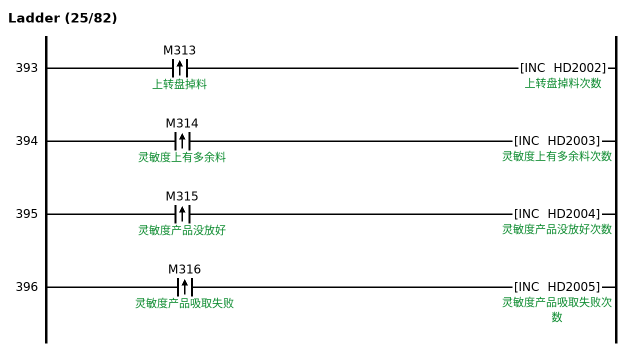
[picture p24: Ladder rows 393-396]
LDP    M313	; 上转盘掉料
INC    HD2002	; 上转盘掉料次数
LDP    M314	; 灵敏度上有多余料
INC    HD2003	; 灵敏度上有多余料次数
LDP    M315	; 灵敏度产品没放好
INC    HD2004	; 灵敏度产品没放好次数
LDP    M316	; 灵敏度产品吸取失败
INC    HD2005	; 灵敏度产品吸取失败次数

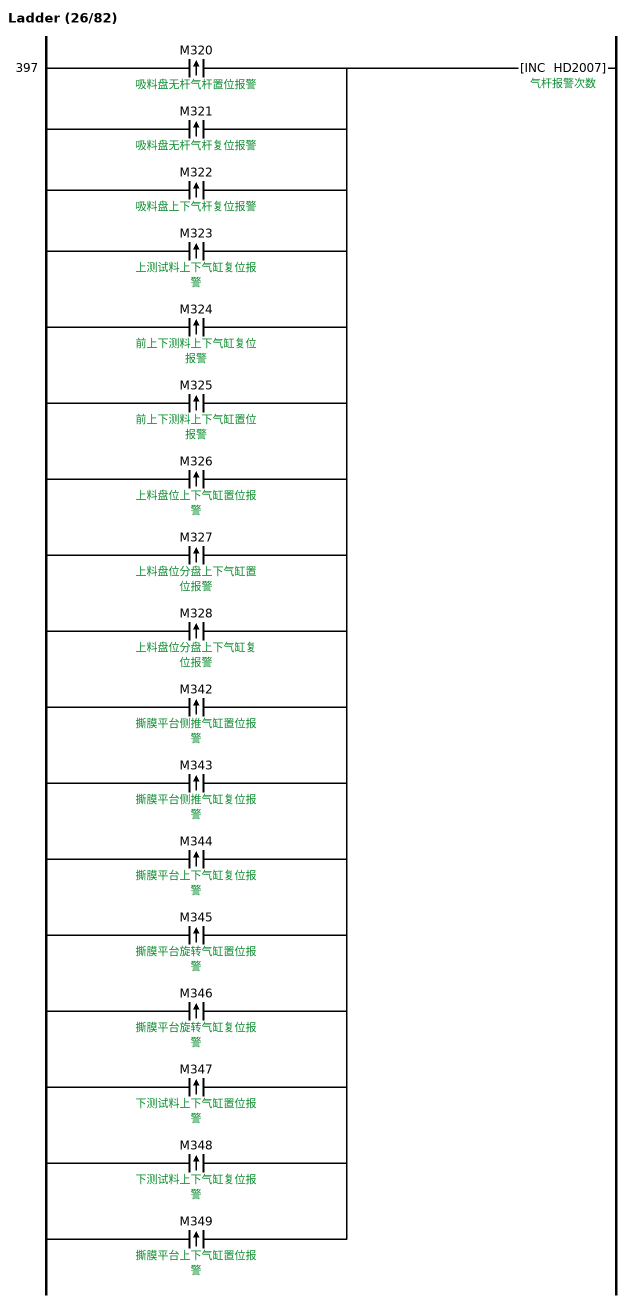
LDP    M320	; 吸料盘无杆气杆置位报警
ORP    M321	; 吸料盘无杆气杆复位报警
ORP    M322	; 吸料盘上下气杆复位报警
ORP    M323	; 上测试料上下气缸复位报警
ORP    M324	; 前上下测料上下气缸复位报警
ORP    M325	; 前上下测料上下气缸置位报警
ORP    M326	; 上料盘位上下气缸置位报警
ORP    M327	; 上料盘位分盘上下气缸置位报警
ORP    M328	; 上料盘位分盘上下气缸复位报警
ORP    M342	; 撕膜平台侧推气缸置位报警
ORP    M343	; 撕膜平台侧推气缸复位报警
ORP    M344	; 撕膜平台上下气缸复位报警
ORP    M345	; 撕膜平台旋转气缸置位报警
ORP    M346	; 撕膜平台旋转气缸复位报警
ORP    M347	; 下测试料上下气缸置位报警
ORP    M348	; 下测试料上下气缸复位报警
ORP    M349	; 撕膜平台上下气缸置位报警
INC    HD2007	; 气杆报警次数

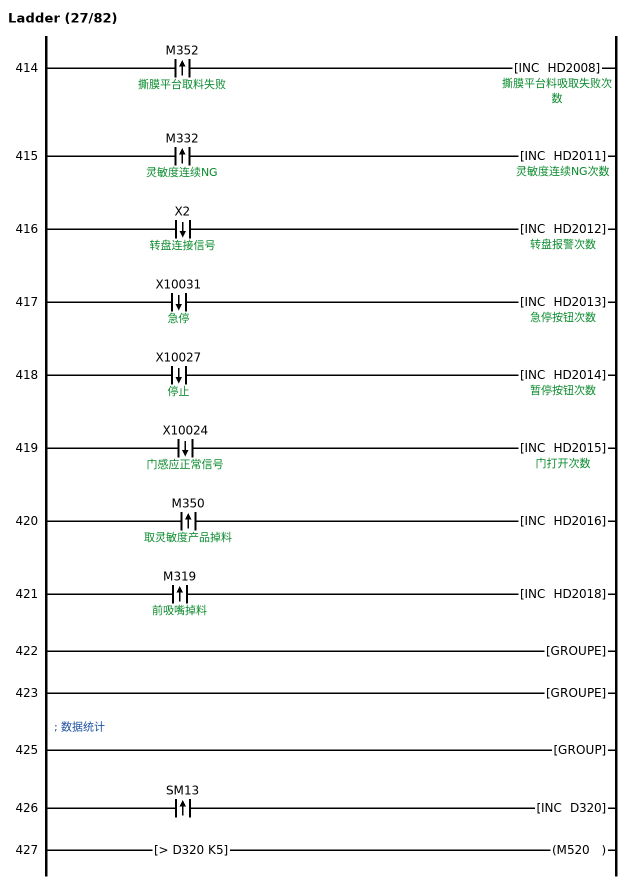
LDP    M352	; 撕膜平台取料失败
INC    HD2008	; 撕膜平台料吸取失败次数
LDP    M332	; 灵敏度连续NG
INC    HD2011	; 灵敏度连续NG次数
LDF    X2	; 转盘连接信号
INC    HD2012	; 转盘报警次数
LDF    X10031	; 急停
INC    HD2013	; 急停按钮次数
LDF    X10027	; 停止
INC    HD2014	; 暂停按钮次数
LDF    X10024	; 门感应正常信号
INC    HD2015	; 门打开次数
LDP    M350	; 取灵敏度产品掉料
INC    HD2016
LDP    M319	; 前吸嘴掉料
INC    HD2018
GROUPE
GROUPE
; 数据统计
GROUP
LDP    SM13
INC    D320
LD>    D320 K5
OUT    M520

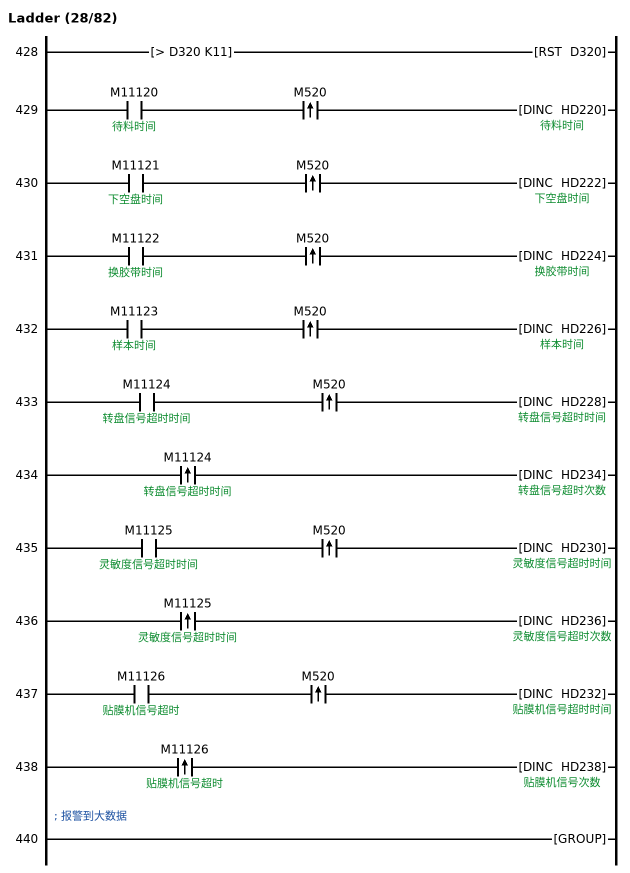
LD>    D320 K11
RST    D320
LD     M11120	; 待料时间
ANDP   M520
DINC   HD220	; 待料时间
LD     M11121	; 下空盘时间
ANDP   M520
DINC   HD222	; 下空盘时间
LD     M11122	; 换胶带时间
ANDP   M520
DINC   HD224	; 换胶带时间
LD     M11123	; 样本时间
ANDP   M520
DINC   HD226	; 样本时间
LD     M11124	; 转盘信号超时时间
ANDP   M520
DINC   HD228	; 转盘信号超时时间
LDP    M11124	; 转盘信号超时时间
DINC   HD234	; 转盘信号超时次数
LD     M11125	; 灵敏度信号超时时间
ANDP   M520
DINC   HD230	; 灵敏度信号超时时间
LDP    M11125	; 灵敏度信号超时时间
DINC   HD236	; 灵敏度信号超时次数
LD     M11126	; 贴膜机信号超时
ANDP   M520
DINC   HD232	; 贴膜机信号超时时间
LDP    M11126	; 贴膜机信号超时
DINC   HD238	; 贴膜机信号次数
; 报警到大数据
GROUP

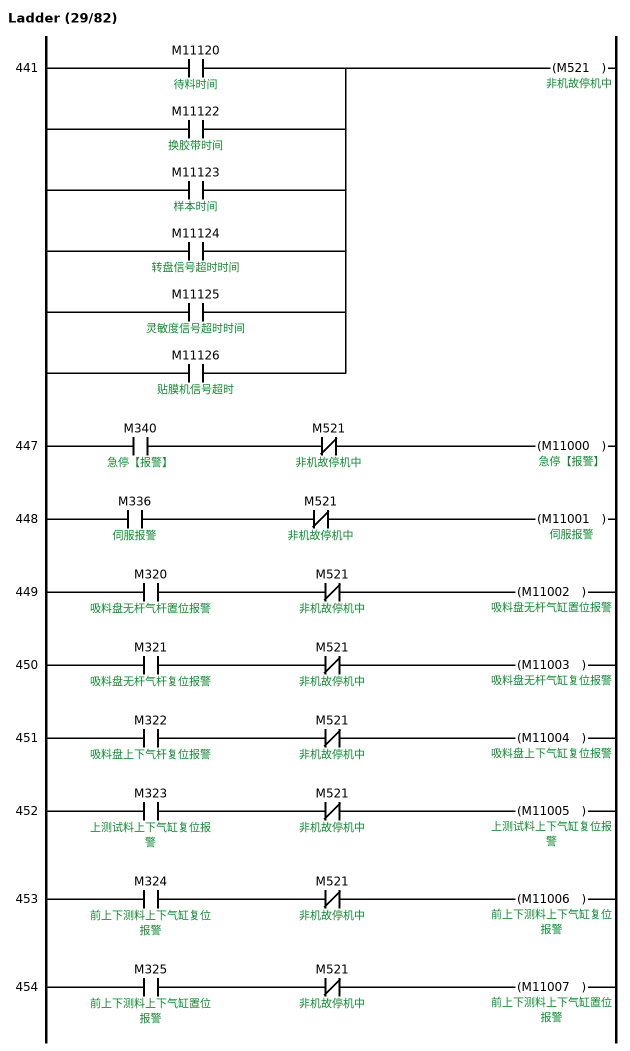
LD     M11120	; 待料时间
OR     M11122	; 换胶带时间
OR     M11123	; 样本时间
OR     M11124	; 转盘信号超时时间
OR     M11125	; 灵敏度信号超时时间
OR     M11126	; 贴膜机信号超时
OUT    M521	; 非机故停机中
LD     M340	; 急停【报警】
ANI    M521	; 非机故停机中
OUT    M11000	; 急停【报警】
LD     M336	; 伺服报警
ANI    M521	; 非机故停机中
OUT    M11001	; 伺服报警
LD     M320	; 吸料盘无杆气杆置位报警
ANI    M521	; 非机故停机中
OUT    M11002	; 吸料盘无杆气缸置位报警
LD     M321	; 吸料盘无杆气杆复位报警
ANI    M521	; 非机故停机中
OUT    M11003	; 吸料盘无杆气缸复位报警
LD     M322	; 吸料盘上下气杆复位报警
ANI    M521	; 非机故停机中
OUT    M11004	; 吸料盘上下气缸复位报警
LD     M323	; 上测试料上下气缸复位报警
ANI    M521	; 非机故停机中
OUT    M11005	; 上测试料上下气缸复位报警
LD     M324	; 前上下测料上下气缸复位报警
ANI    M521	; 非机故停机中
OUT    M11006	; 前上下测料上下气缸复位报警
LD     M325	; 前上下测料上下气缸置位报警
ANI    M521	; 非机故停机中
OUT    M11007	; 前上下测料上下气缸置位报警

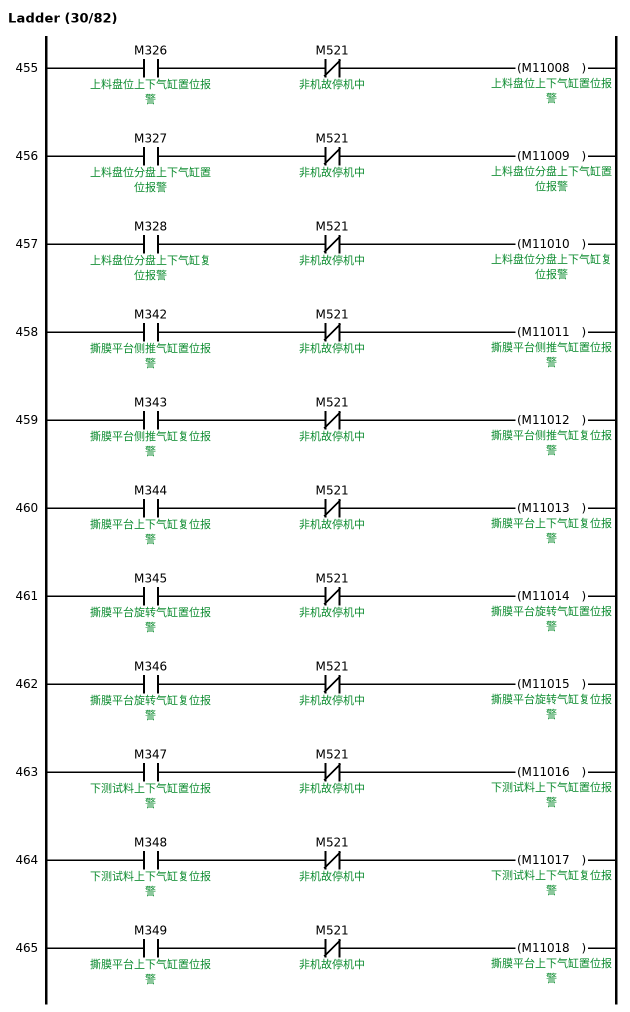
LD     M326	; 上料盘位上下气缸置位报警
ANI    M521	; 非机故停机中
OUT    M11008	; 上料盘位上下气缸置位报警
LD     M327	; 上料盘位分盘上下气缸置位报警
ANI    M521	; 非机故停机中
OUT    M11009	; 上料盘位分盘上下气缸置位报警
LD     M328	; 上料盘位分盘上下气缸复位报警
ANI    M521	; 非机故停机中
OUT    M11010	; 上料盘位分盘上下气缸复位报警
LD     M342	; 撕膜平台侧推气缸置位报警
ANI    M521	; 非机故停机中
OUT    M11011	; 撕膜平台侧推气缸置位报警
LD     M343	; 撕膜平台侧推气缸复位报警
ANI    M521	; 非机故停机中
OUT    M11012	; 撕膜平台侧推气缸复位报警
LD     M344	; 撕膜平台上下气缸复位报警
ANI    M521	; 非机故停机中
OUT    M11013	; 撕膜平台上下气缸复位报警
LD     M345	; 撕膜平台旋转气缸置位报警
ANI    M521	; 非机故停机中
OUT    M11014	; 撕膜平台旋转气缸置位报警
LD     M346	; 撕膜平台旋转气缸复位报警
ANI    M521	; 非机故停机中
OUT    M11015	; 撕膜平台旋转气缸复位报警
LD     M347	; 下测试料上下气缸置位报警
ANI    M521	; 非机故停机中
OUT    M11016	; 下测试料上下气缸置位报警
LD     M348	; 下测试料上下气缸复位报警
ANI    M521	; 非机故停机中
OUT    M11017	; 下测试料上下气缸复位报警
LD     M349	; 撕膜平台上下气缸置位报警
ANI    M521	; 非机故停机中
OUT    M11018	; 撕膜平台上下气缸置位报警

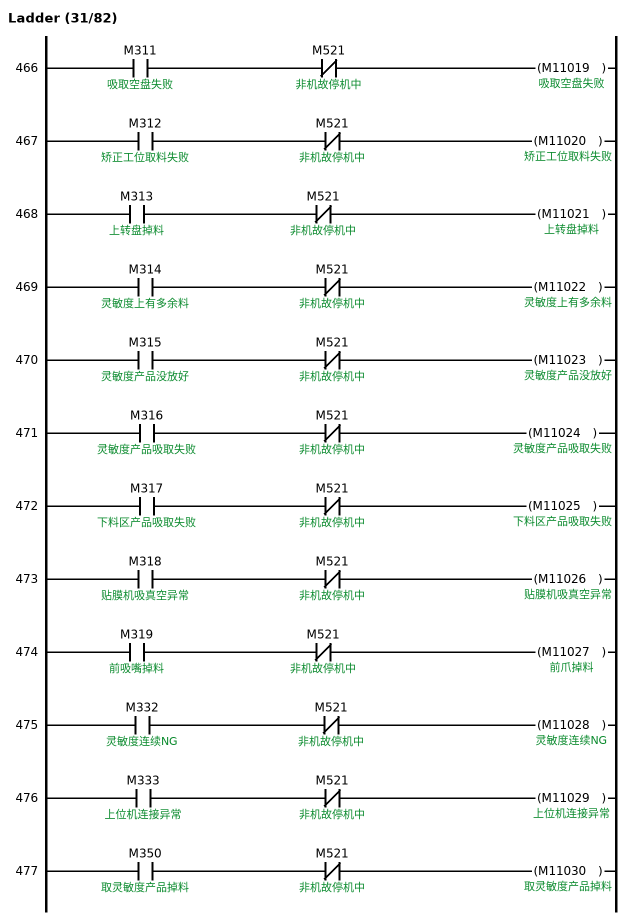
LD     M311	; 吸取空盘失败
ANI    M521	; 非机故停机中
OUT    M11019	; 吸取空盘失败
LD     M312	; 矫正工位取料失败
ANI    M521	; 非机故停机中
OUT    M11020	; 矫正工位取料失败
LD     M313	; 上转盘掉料
ANI    M521	; 非机故停机中
OUT    M11021	; 上转盘掉料
LD     M314	; 灵敏度上有多余料
ANI    M521	; 非机故停机中
OUT    M11022	; 灵敏度上有多余料
LD     M315	; 灵敏度产品没放好
ANI    M521	; 非机故停机中
OUT    M11023	; 灵敏度产品没放好
LD     M316	; 灵敏度产品吸取失败
ANI    M521	; 非机故停机中
OUT    M11024	; 灵敏度产品吸取失败
LD     M317	; 下料区产品吸取失败
ANI    M521	; 非机故停机中
OUT    M11025	; 下料区产品吸取失败
LD     M318	; 贴膜机吸真空异常
ANI    M521	; 非机故停机中
OUT    M11026	; 贴膜机吸真空异常
LD     M319	; 前吸嘴掉料
ANI    M521	; 非机故停机中
OUT    M11027	; 前爪掉料
LD     M332	; 灵敏度连续NG
ANI    M521	; 非机故停机中
OUT    M11028	; 灵敏度连续NG
LD     M333	; 上位机连接异常
ANI    M521	; 非机故停机中
OUT    M11029	; 上位机连接异常
LD     M350	; 取灵敏度产品掉料
ANI    M521	; 非机故停机中
OUT    M11030	; 取灵敏度产品掉料

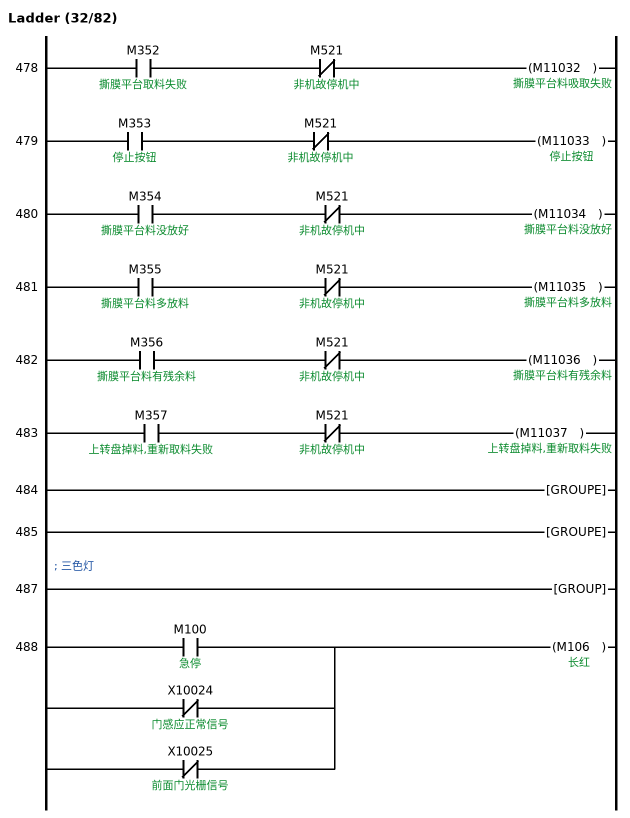
LD     M352	; 撕膜平台取料失败
ANI    M521	; 非机故停机中
OUT    M11032	; 撕膜平台料吸取失败
LD     M353	; 停止按钮
ANI    M521	; 非机故停机中
OUT    M11033	; 停止按钮
LD     M354	; 撕膜平台料没放好
ANI    M521	; 非机故停机中
OUT    M11034	; 撕膜平台料没放好
LD     M355	; 撕膜平台料多放料
ANI    M521	; 非机故停机中
OUT    M11035	; 撕膜平台料多放料
LD     M356	; 撕膜平台料有残余料
ANI    M521	; 非机故停机中
OUT    M11036	; 撕膜平台料有残余料
LD     M357	; 上转盘掉料,重新取料失败
ANI    M521	; 非机故停机中
OUT    M11037	; 上转盘掉料,重新取料失败
GROUPE
GROUPE
; 三色灯
GROUP
LD     M100	; 急停
ORI    X10024	; 门感应正常信号
ORI    X10025	; 前面门光栅信号
OUT    M106	; 长红

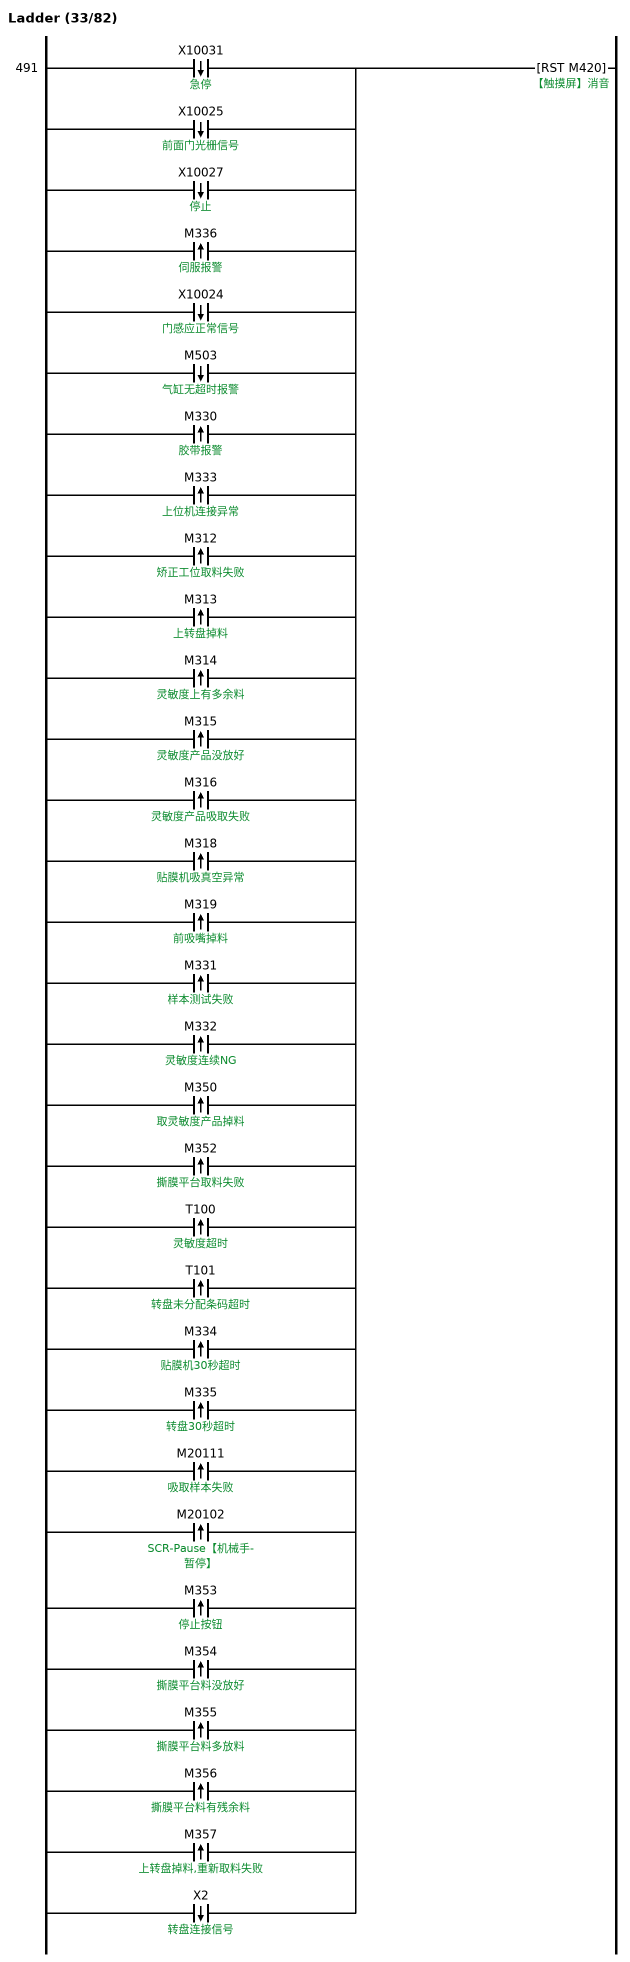
LDF    X10031	; 急停
ORF    X10025	; 前面门光栅信号
ORF    X10027	; 停止
ORP    M336	; 伺服报警
ORF    X10024	; 门感应正常信号
ORF    M503	; 气缸无超时报警
ORP    M330	; 胶带报警
ORP    M333	; 上位机连接异常
ORP    M312	; 矫正工位取料失败
ORP    M313	; 上转盘掉料
ORP    M314	; 灵敏度上有多余料
ORP    M315	; 灵敏度产品没放好
ORP    M316	; 灵敏度产品吸取失败
ORP    M318	; 贴膜机吸真空异常
ORP    M319	; 前吸嘴掉料
ORP    M331	; 样本测试失败
ORP    M332	; 灵敏度连续NG
ORP    M350	; 取灵敏度产品掉料
ORP    M352	; 撕膜平台取料失败
ORP    T100	; 灵敏度超时
ORP    T101	; 转盘未分配条码超时
ORP    M334	; 贴膜机30秒超时
ORP    M335	; 转盘30秒超时
ORP    M20111	; 吸取样本失败
ORP    M20102	; SCR-Pause【机械手-暂停】
ORP    M353	; 停止按钮
ORP    M354	; 撕膜平台料没放好
ORP    M355	; 撕膜平台料多放料
ORP    M356	; 撕膜平台料有残余料
ORP    M357	; 上转盘掉料,重新取料失败
ORF    X2	; 转盘连接信号
RST    M420	; 【触摸屏】消音

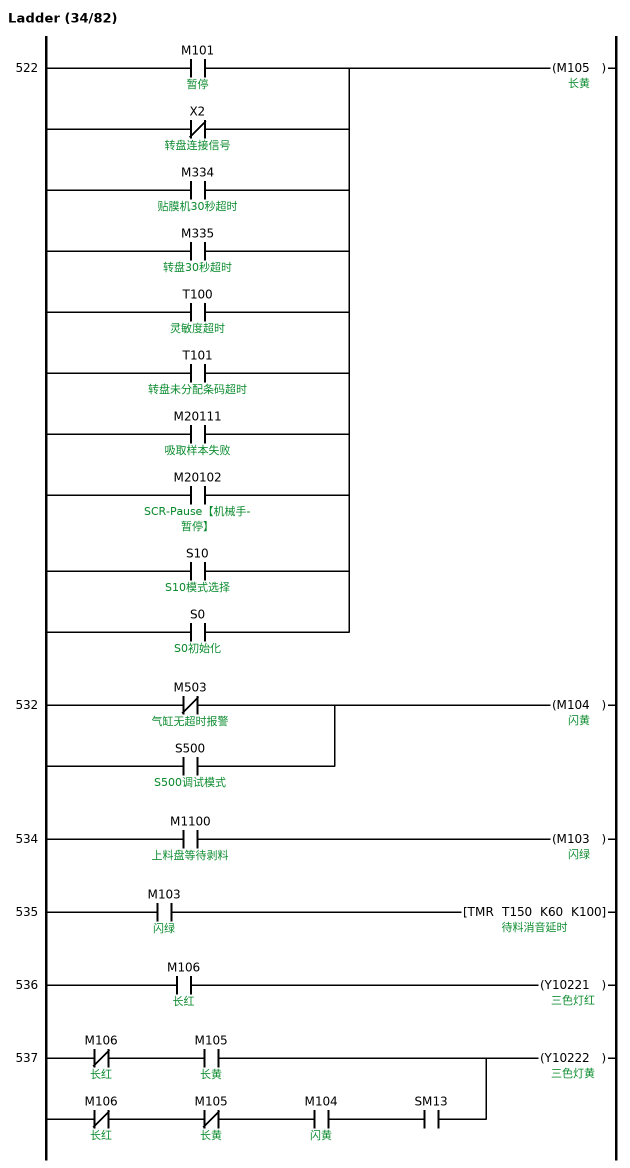
LD     M101	; 暂停
ORI    X2	; 转盘连接信号
OR     M334	; 贴膜机30秒超时
OR     M335	; 转盘30秒超时
OR     T100	; 灵敏度超时
OR     T101	; 转盘未分配条码超时
OR     M20111	; 吸取样本失败
OR     M20102	; SCR-Pause【机械手-暂停】
OR     S10	; S10模式选择
OR     S0	; S0初始化
OUT    M105	; 长黄
LDI    M503	; 气缸无超时报警
OR     S500	; S500调试模式
OUT    M104	; 闪黄
LD     M1100	; 上料盘等待剥料
OUT    M103	; 闪绿
LD     M103	; 闪绿
TMR    T150 K60 K100	; 待料消音延时
LD     M106	; 长红
OUT    Y10221	; 三色灯红
LDI    M106	; 长红
AND    M105	; 长黄
LDI    M106	; 长红
ANI    M105	; 长黄
AND    M104	; 闪黄
AND    SM13
ORB
OUT    Y10222	; 三色灯黄

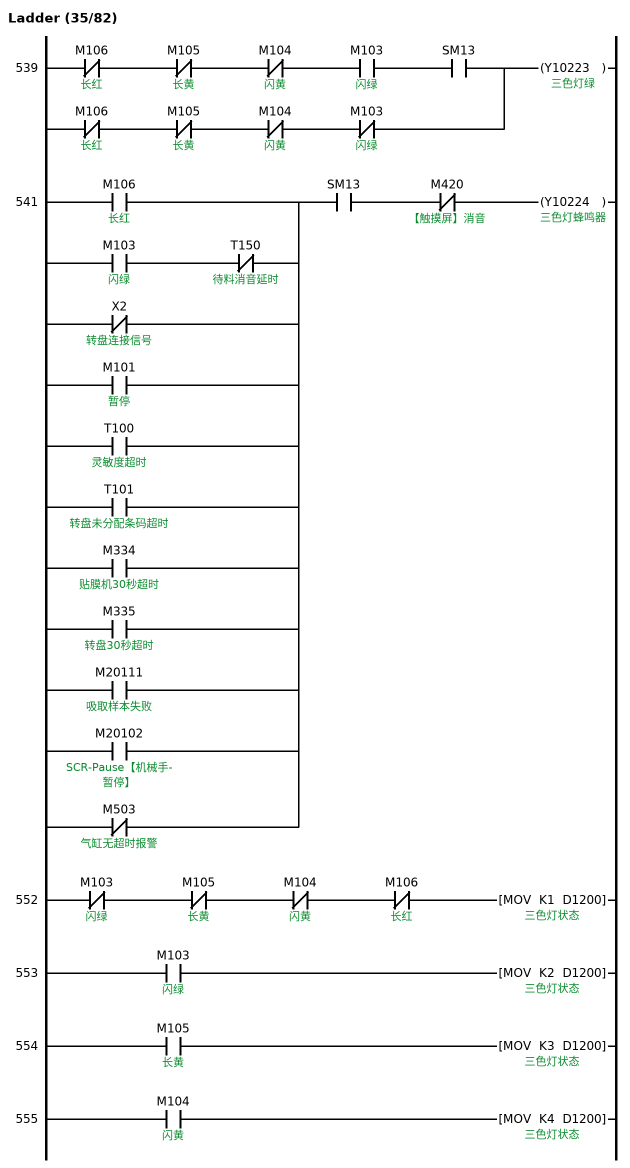
LDI    M106	; 长红
ANI    M105	; 长黄
ANI    M104	; 闪黄
AND    M103	; 闪绿
AND    SM13
LDI    M106	; 长红
ANI    M105	; 长黄
ANI    M104	; 闪黄
ANI    M103	; 闪绿
ORB
OUT    Y10223	; 三色灯绿
LD     M106	; 长红
LD     M103	; 闪绿
ANI    T150	; 待料消音延时
ORB
ORI    X2	; 转盘连接信号
OR     M101	; 暂停
OR     T100	; 灵敏度超时
OR     T101	; 转盘未分配条码超时
OR     M334	; 贴膜机30秒超时
OR     M335	; 转盘30秒超时
OR     M20111	; 吸取样本失败
OR     M20102	; SCR-Pause【机械手-暂停】
ORI    M503	; 气缸无超时报警
AND    SM13
ANI    M420	; 【触摸屏】消音
OUT    Y10224	; 三色灯蜂鸣器
LDI    M103	; 闪绿
ANI    M105	; 长黄
ANI    M104	; 闪黄
ANI    M106	; 长红
MOV    K1 D1200	; 三色灯状态
LD     M103	; 闪绿
MOV    K2 D1200	; 三色灯状态
LD     M105	; 长黄
MOV    K3 D1200	; 三色灯状态
LD     M104	; 闪黄
MOV    K4 D1200	; 三色灯状态

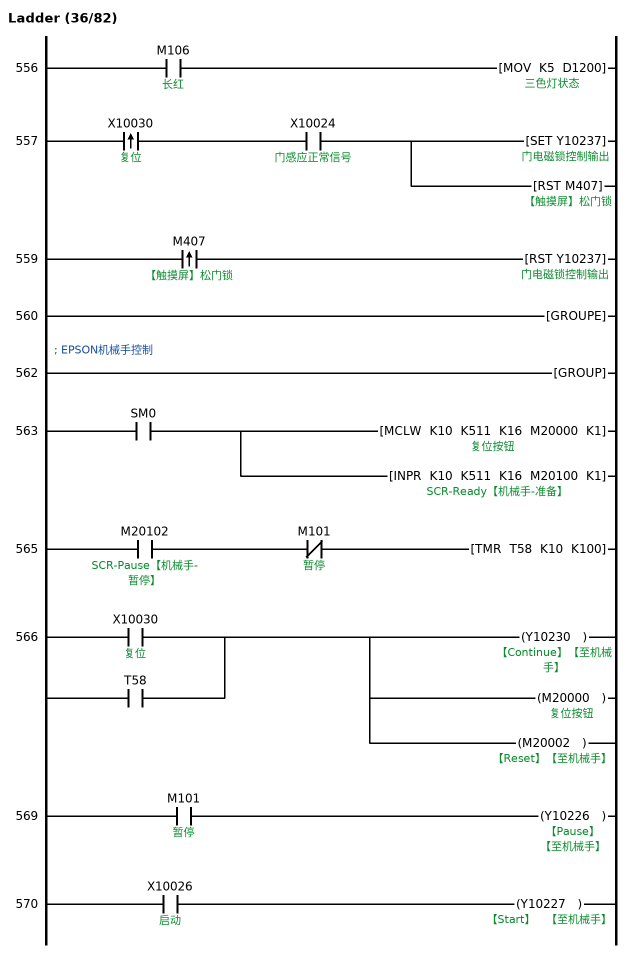
LD     M106	; 长红
MOV    K5 D1200	; 三色灯状态
LDP    X10030	; 复位
AND    X10024	; 门感应正常信号
SET    Y10237	; 门电磁锁控制输出
RST    M407	; 【触摸屏】松门锁
LDP    M407	; 【触摸屏】松门锁
RST    Y10237	; 门电磁锁控制输出
GROUPE
; EPSON机械手控制
GROUP
LD     SM0
MCLW   K10 K511 K16 M20000 K1	; 复位按钮
INPR   K10 K511 K16 M20100 K1	; SCR-Ready【机械手-准备】
LD     M20102	; SCR-Pause【机械手-暂停】
ANI    M101	; 暂停
TMR    T58 K10 K100
LD     X10030	; 复位
OR     T58
OUT    Y10230	; 【Continue】【至机械手】
OUT    M20000	; 复位按钮
OUT    M20002	; 【Reset】【至机械手】
LD     M101	; 暂停
OUT    Y10226	; 【Pause】   【至机械手】
LD     X10026	; 启动
OUT    Y10227	; 【Start】   【至机械手】

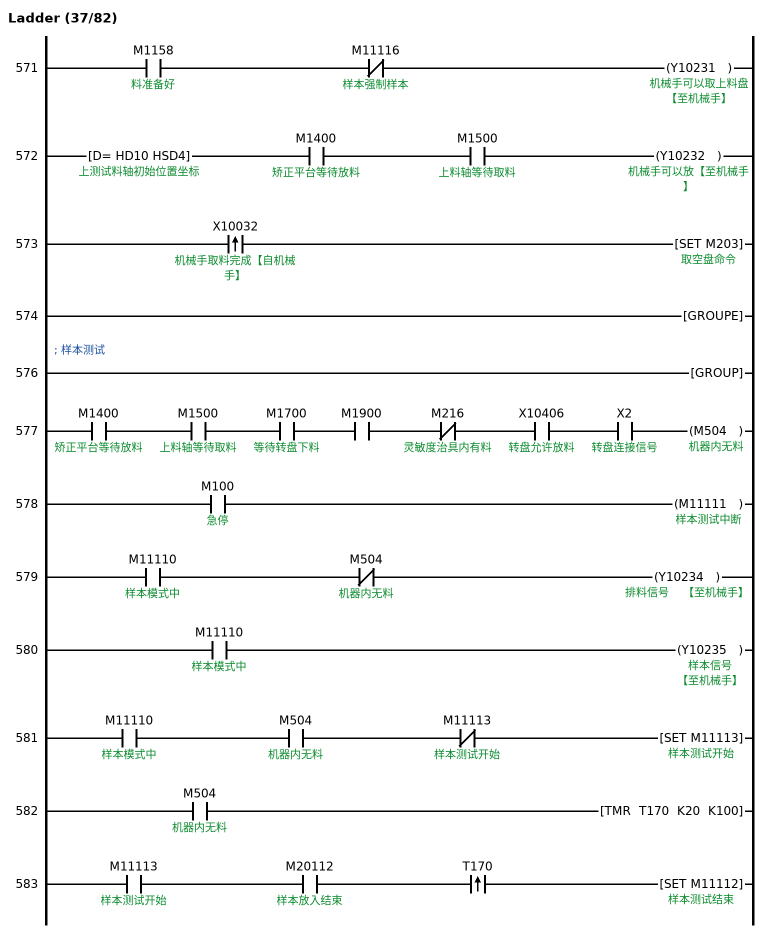
LD     M1158	; 料准备好
ANI    M11116	; 样本强制样本
OUT    Y10231	; 机械手可以取上料盘  【至机械手】
DLD=   HD10 HSD4	; 上测试料轴初始位置坐标
AND    M1400	; 矫正平台等待放料
AND    M1500	; 上料轴等待取料
OUT    Y10232	; 机械手可以放【至机械手】
LDP    X10032	; 机械手取料完成【自机械手】
SET    M203	; 取空盘命令
GROUPE
; 样本测试
GROUP
LD     M1400	; 矫正平台等待放料
AND    M1500	; 上料轴等待取料
AND    M1700	; 等待转盘下料
AND    M1900
ANI    M216	; 灵敏度治具内有料
AND    X10406	; 转盘允许放料
AND    X2	; 转盘连接信号
OUT    M504	; 机器内无料
LD     M100	; 急停
OUT    M11111	; 样本测试中断
LD     M11110	; 样本模式中
ANI    M504	; 机器内无料
OUT    Y10234	; 排料信号    【至机械手】
LD     M11110	; 样本模式中
OUT    Y10235	; 样本信号     【至机械手】
LD     M11110	; 样本模式中
AND    M504	; 机器内无料
ANI    M11113	; 样本测试开始
SET    M11113	; 样本测试开始
LD     M504	; 机器内无料
TMR    T170 K20 K100
LD     M11113	; 样本测试开始
AND    M20112	; 样本放入结束
ANDP   T170
SET    M11112	; 样本测试结束

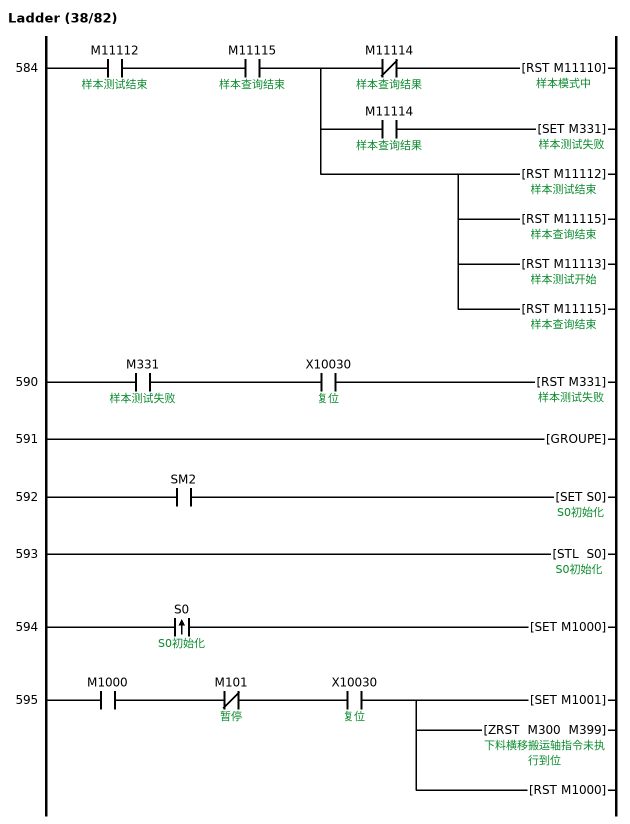
LD     M11112	; 样本测试结束
AND    M11115	; 样本查询结束
MPS
ANI    M11114	; 样本查询结果
RST    M11110	; 样本模式中
MRD
AND    M11114	; 样本查询结果
SET    M331	; 样本测试失败
MPP
RST    M11112	; 样本测试结束
RST    M11115	; 样本查询结束
RST    M11113	; 样本测试开始
RST    M11115	; 样本查询结束
LD     M331	; 样本测试失败
AND    X10030	; 复位
RST    M331	; 样本测试失败
GROUPE
LD     SM2
SET    S0	; S0初始化
STL    S0	; S0初始化
LDP    S0	; S0初始化
SET    M1000
LD     M1000
ANI    M101	; 暂停
AND    X10030	; 复位
SET    M1001
ZRST   M300 M399	; 下料横移搬运轴指令未执行到位
RST    M1000

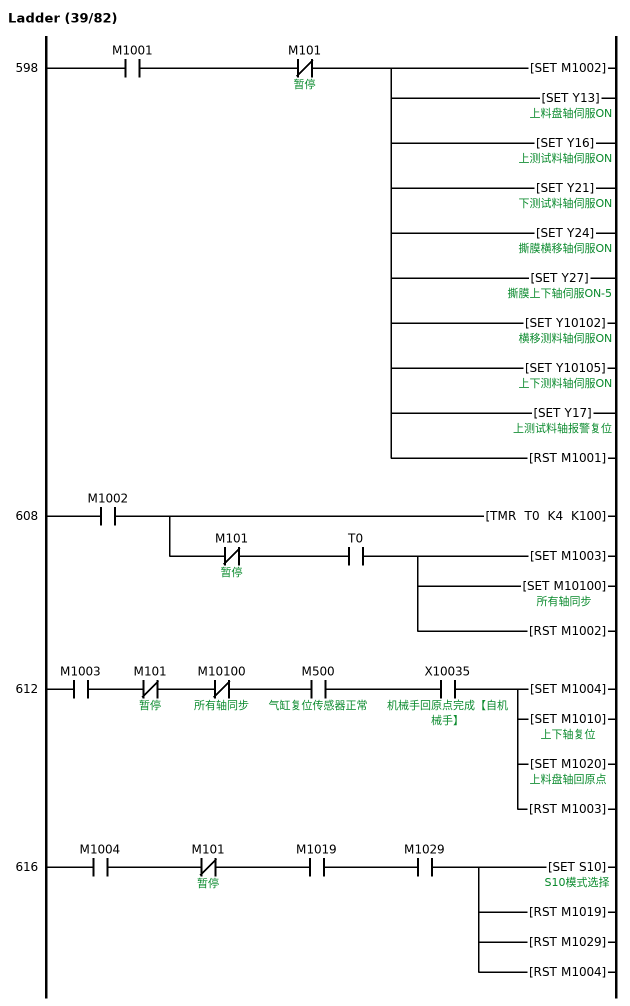
LD     M1001
ANI    M101	; 暂停
SET    M1002
SET    Y13	; 上料盘轴伺服ON
SET    Y16	; 上测试料轴伺服ON
SET    Y21	; 下测试料轴伺服ON
SET    Y24	; 撕膜横移轴伺服ON
SET    Y27	; 撕膜上下轴伺服ON-5
SET    Y10102	; 横移测料轴伺服ON
SET    Y10105	; 上下测料轴伺服ON
SET    Y17	; 上测试料轴报警复位
RST    M1001
LD     M1002
TMR    T0 K4 K100
ANI    M101	; 暂停
AND    T0
SET    M1003
SET    M10100	; 所有轴同步
RST    M1002
LD     M1003
ANI    M101	; 暂停
ANI    M10100	; 所有轴同步
AND    M500	; 气缸复位传感器正常
AND    X10035	; 机械手回原点完成【自机械手】
SET    M1004
SET    M1010	; 上下轴复位
SET    M1020	; 上料盘轴回原点
RST    M1003
LD     M1004
ANI    M101	; 暂停
AND    M1019
AND    M1029
SET    S10	; S10模式选择
RST    M1019
RST    M1029
RST    M1004

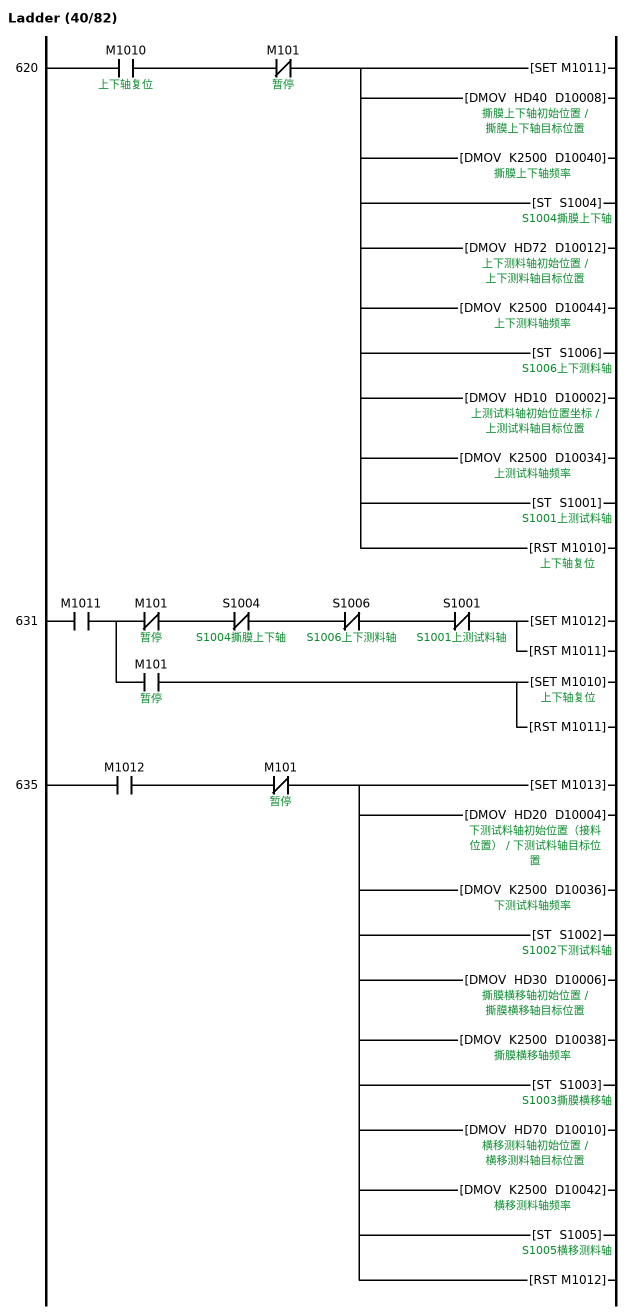
LD     M1010	; 上下轴复位
ANI    M101	; 暂停
SET    M1011
DMOV   HD40 D10008	; 撕膜上下轴初始位置 / 撕膜上下轴目标位置
DMOV   K2500 D10040	; 撕膜上下轴频率
ST     S1004	; S1004撕膜上下轴
DMOV   HD72 D10012	; 上下测料轴初始位置 / 上下测料轴目标位置
DMOV   K2500 D10044	; 上下测料轴频率
ST     S1006	; S1006上下测料轴
DMOV   HD10 D10002	; 上测试料轴初始位置坐标 / 上测试料轴目标位置
DMOV   K2500 D10034	; 上测试料轴频率
ST     S1001	; S1001上测试料轴
RST    M1010	; 上下轴复位
LD     M1011
MPS
ANI    M101	; 暂停
ANI    S1004	; S1004撕膜上下轴
ANI    S1006	; S1006上下测料轴
ANI    S1001	; S1001上测试料轴
SET    M1012
RST    M1011
MPP
AND    M101	; 暂停
SET    M1010	; 上下轴复位
RST    M1011
LD     M1012
ANI    M101	; 暂停
SET    M1013
DMOV   HD20 D10004	; 下测试料轴初始位置（接料位置） / 下测试料轴目标位置
DMOV   K2500 D10036	; 下测试料轴频率
ST     S1002	; S1002下测试料轴
DMOV   HD30 D10006	; 撕膜横移轴初始位置 / 撕膜横移轴目标位置
DMOV   K2500 D10038	; 撕膜横移轴频率
ST     S1003	; S1003撕膜横移轴
DMOV   HD70 D10010	; 横移测料轴初始位置 / 横移测料轴目标位置
DMOV   K2500 D10042	; 横移测料轴频率
ST     S1005	; S1005横移测料轴
RST    M1012

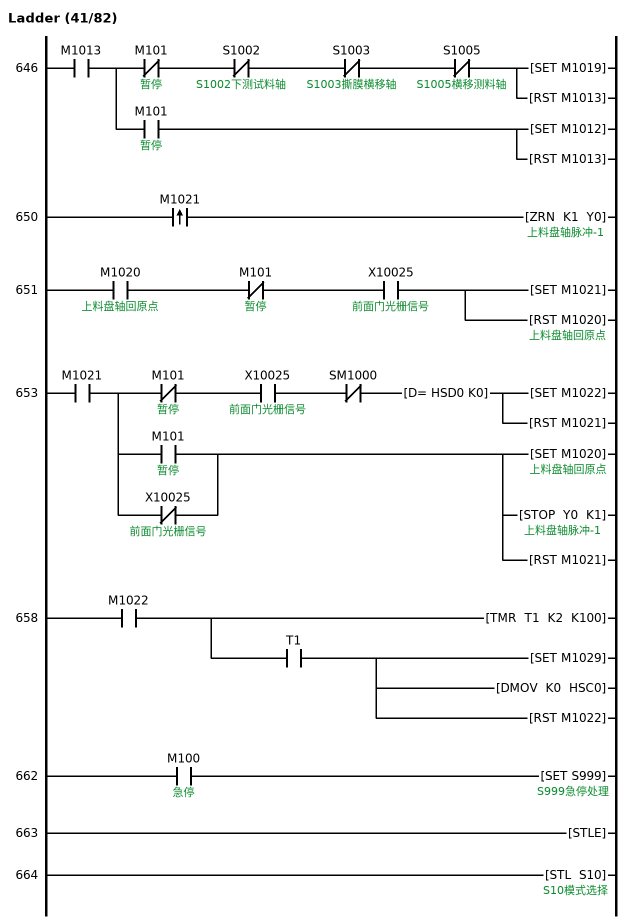
LD     M1013
MPS
ANI    M101	; 暂停
ANI    S1002	; S1002下测试料轴
ANI    S1003	; S1003撕膜横移轴
ANI    S1005	; S1005横移测料轴
SET    M1019
RST    M1013
MPP
AND    M101	; 暂停
SET    M1012
RST    M1013
LDP    M1021
ZRN    K1 Y0	; 上料盘轴脉冲-1
LD     M1020	; 上料盘轴回原点
ANI    M101	; 暂停
AND    X10025	; 前面门光栅信号
SET    M1021
RST    M1020	; 上料盘轴回原点
LD     M1021
MPS
ANI    M101	; 暂停
AND    X10025	; 前面门光栅信号
ANI    SM1000
DAND=  HSD0 K0
SET    M1022
RST    M1021
MPP
LD     M101	; 暂停
ORI    X10025	; 前面门光栅信号
ANB
SET    M1020	; 上料盘轴回原点
STOP   Y0 K1	; 上料盘轴脉冲-1
RST    M1021
LD     M1022
TMR    T1 K2 K100
AND    T1
SET    M1029
DMOV   K0 HSC0
RST    M1022
LD     M100	; 急停
SET    S999	; S999急停处理
STLE
STL    S10	; S10模式选择

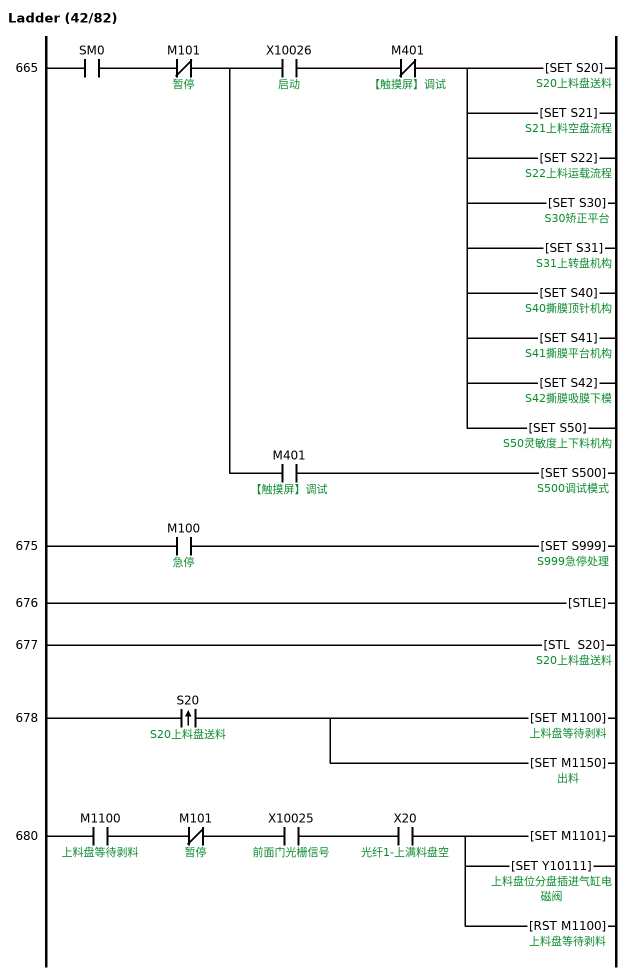
LD     SM0
ANI    M101	; 暂停
MPS
AND    X10026	; 启动
ANI    M401	; 【触摸屏】调试
SET    S20	; S20上料盘送料
SET    S21	; S21上料空盘流程
SET    S22	; S22上料运载流程
SET    S30	; S30矫正平台
SET    S31	; S31上转盘机构
SET    S40	; S40撕膜顶针机构
SET    S41	; S41撕膜平台机构
SET    S42	; S42撕膜吸膜下模
SET    S50	; S50灵敏度上下料机构
MPP
AND    M401	; 【触摸屏】调试
SET    S500	; S500调试模式
LD     M100	; 急停
SET    S999	; S999急停处理
STLE
STL    S20	; S20上料盘送料
LDP    S20	; S20上料盘送料
SET    M1100	; 上料盘等待剥料
SET    M1150	; 出料
LD     M1100	; 上料盘等待剥料
ANI    M101	; 暂停
AND    X10025	; 前面门光栅信号
AND    X20	; 光纤1-上满料盘空
SET    M1101
SET    Y10111	; 上料盘位分盘插进气缸电磁阀
RST    M1100	; 上料盘等待剥料

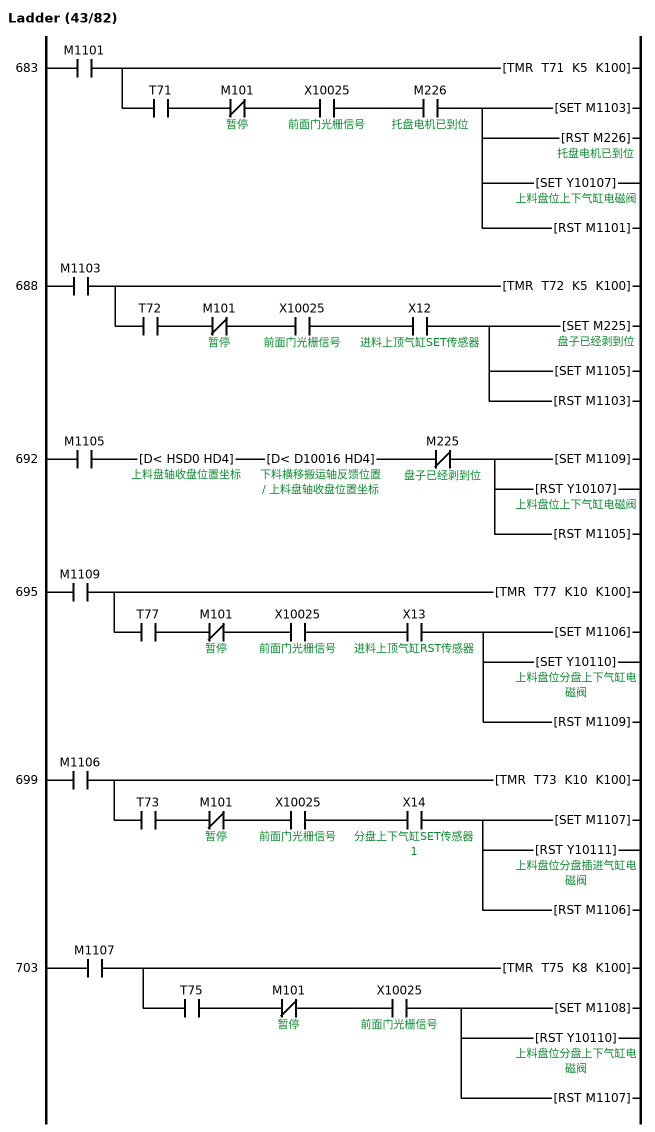
LD     M1101
TMR    T71 K5 K100
AND    T71
ANI    M101	; 暂停
AND    X10025	; 前面门光栅信号
AND    M226	; 托盘电机已到位
SET    M1103
RST    M226	; 托盘电机已到位
SET    Y10107	; 上料盘位上下气缸电磁阀
RST    M1101
LD     M1103
TMR    T72 K5 K100
AND    T72
ANI    M101	; 暂停
AND    X10025	; 前面门光栅信号
AND    X12	; 进料上顶气缸SET传感器
SET    M225	; 盘子已经剥到位
SET    M1105
RST    M1103
LD     M1105
DAND<  HSD0 HD4	; 上料盘轴收盘位置坐标
DAND<  D10016 HD4	; 下料横移搬运轴反馈位置 / 上料盘轴收盘位置坐标
ANI    M225	; 盘子已经剥到位
SET    M1109
RST    Y10107	; 上料盘位上下气缸电磁阀
RST    M1105
LD     M1109
TMR    T77 K10 K100
AND    T77
ANI    M101	; 暂停
AND    X10025	; 前面门光栅信号
AND    X13	; 进料上顶气缸RST传感器
SET    M1106
SET    Y10110	; 上料盘位分盘上下气缸电磁阀
RST    M1109
LD     M1106
TMR    T73 K10 K100
AND    T73
ANI    M101	; 暂停
AND    X10025	; 前面门光栅信号
AND    X14	; 分盘上下气缸SET传感器1
SET    M1107
RST    Y10111	; 上料盘位分盘插进气缸电磁阀
RST    M1106
LD     M1107
TMR    T75 K8 K100
AND    T75
ANI    M101	; 暂停
AND    X10025	; 前面门光栅信号
SET    M1108
RST    Y10110	; 上料盘位分盘上下气缸电磁阀
RST    M1107

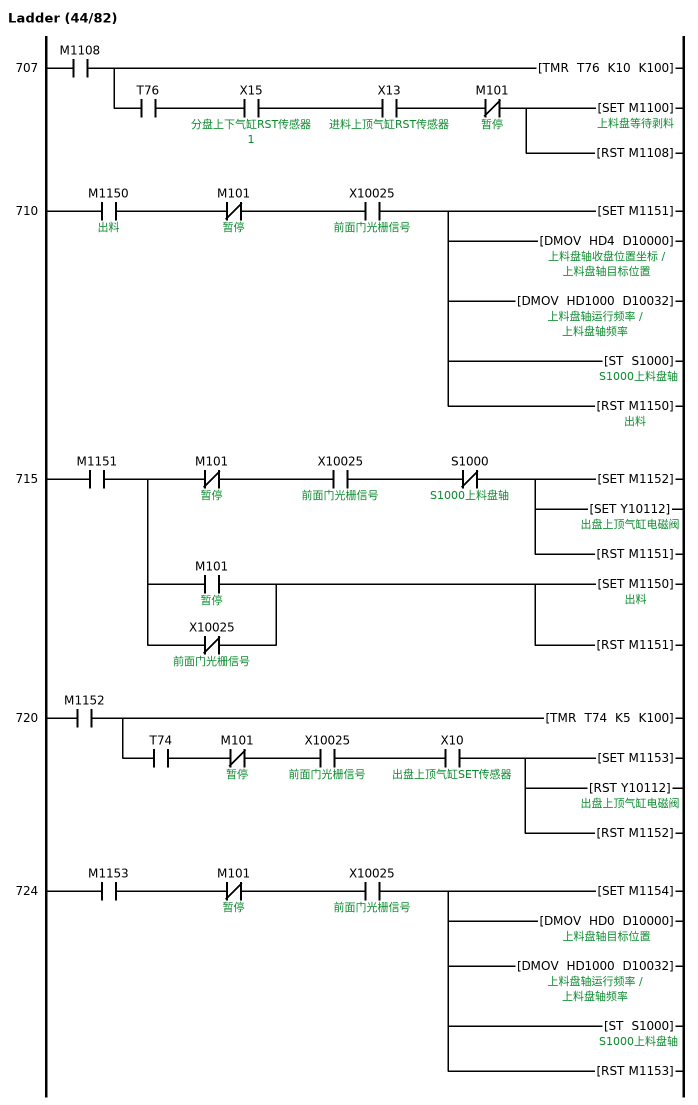
LD     M1108
TMR    T76 K10 K100
AND    T76
AND    X15	; 分盘上下气缸RST传感器1
AND    X13	; 进料上顶气缸RST传感器
ANI    M101	; 暂停
SET    M1100	; 上料盘等待剥料
RST    M1108
LD     M1150	; 出料
ANI    M101	; 暂停
AND    X10025	; 前面门光栅信号
SET    M1151
DMOV   HD4 D10000	; 上料盘轴收盘位置坐标 / 上料盘轴目标位置
DMOV   HD1000 D10032	; 上料盘轴运行频率 / 上料盘轴频率
ST     S1000	; S1000上料盘轴
RST    M1150	; 出料
LD     M1151
MPS
ANI    M101	; 暂停
AND    X10025	; 前面门光栅信号
ANI    S1000	; S1000上料盘轴
SET    M1152
SET    Y10112	; 出盘上顶气缸电磁阀
RST    M1151
MPP
LD     M101	; 暂停
ORI    X10025	; 前面门光栅信号
ANB
SET    M1150	; 出料
RST    M1151
LD     M1152
TMR    T74 K5 K100
AND    T74
ANI    M101	; 暂停
AND    X10025	; 前面门光栅信号
AND    X10	; 出盘上顶气缸SET传感器
SET    M1153
RST    Y10112	; 出盘上顶气缸电磁阀
RST    M1152
LD     M1153
ANI    M101	; 暂停
AND    X10025	; 前面门光栅信号
SET    M1154
DMOV   HD0 D10000	; 上料盘轴目标位置
DMOV   HD1000 D10032	; 上料盘轴运行频率 / 上料盘轴频率
ST     S1000	; S1000上料盘轴
RST    M1153

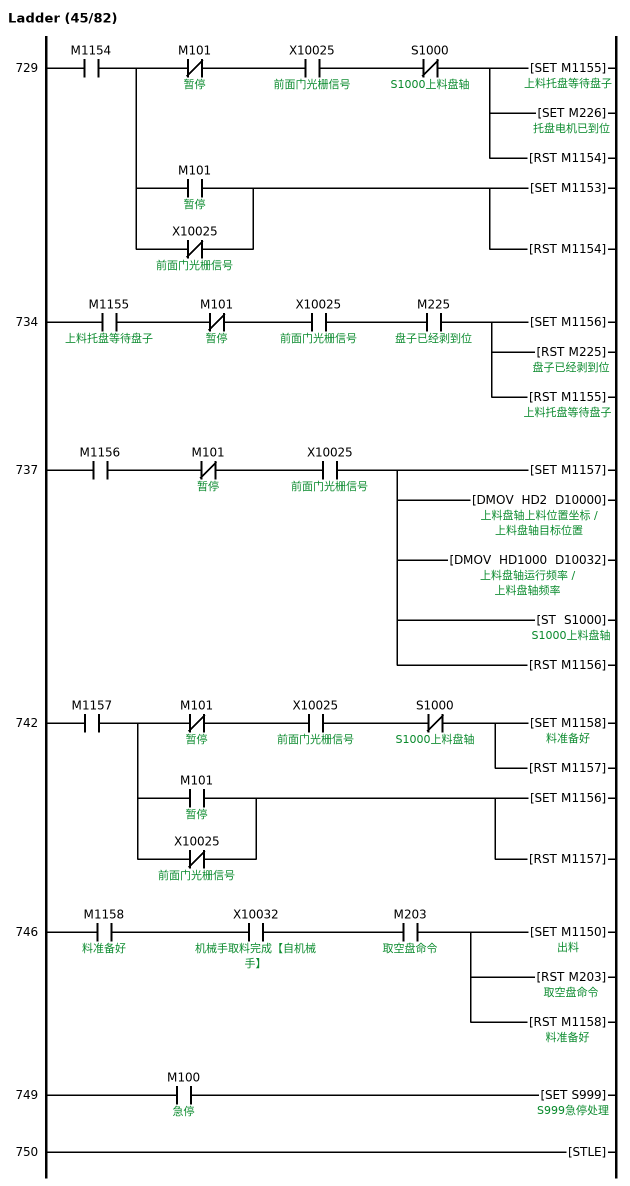
LD     M1154
MPS
ANI    M101	; 暂停
AND    X10025	; 前面门光栅信号
ANI    S1000	; S1000上料盘轴
SET    M1155	; 上料托盘等待盘子
SET    M226	; 托盘电机已到位
RST    M1154
MPP
LD     M101	; 暂停
ORI    X10025	; 前面门光栅信号
ANB
SET    M1153
RST    M1154
LD     M1155	; 上料托盘等待盘子
ANI    M101	; 暂停
AND    X10025	; 前面门光栅信号
AND    M225	; 盘子已经剥到位
SET    M1156
RST    M225	; 盘子已经剥到位
RST    M1155	; 上料托盘等待盘子
LD     M1156
ANI    M101	; 暂停
AND    X10025	; 前面门光栅信号
SET    M1157
DMOV   HD2 D10000	; 上料盘轴上料位置坐标 / 上料盘轴目标位置
DMOV   HD1000 D10032	; 上料盘轴运行频率 / 上料盘轴频率
ST     S1000	; S1000上料盘轴
RST    M1156
LD     M1157
MPS
ANI    M101	; 暂停
AND    X10025	; 前面门光栅信号
ANI    S1000	; S1000上料盘轴
SET    M1158	; 料准备好
RST    M1157
MPP
LD     M101	; 暂停
ORI    X10025	; 前面门光栅信号
ANB
SET    M1156
RST    M1157
LD     M1158	; 料准备好
AND    X10032	; 机械手取料完成【自机械手】
AND    M203	; 取空盘命令
SET    M1150	; 出料
RST    M203	; 取空盘命令
RST    M1158	; 料准备好
LD     M100	; 急停
SET    S999	; S999急停处理
STLE

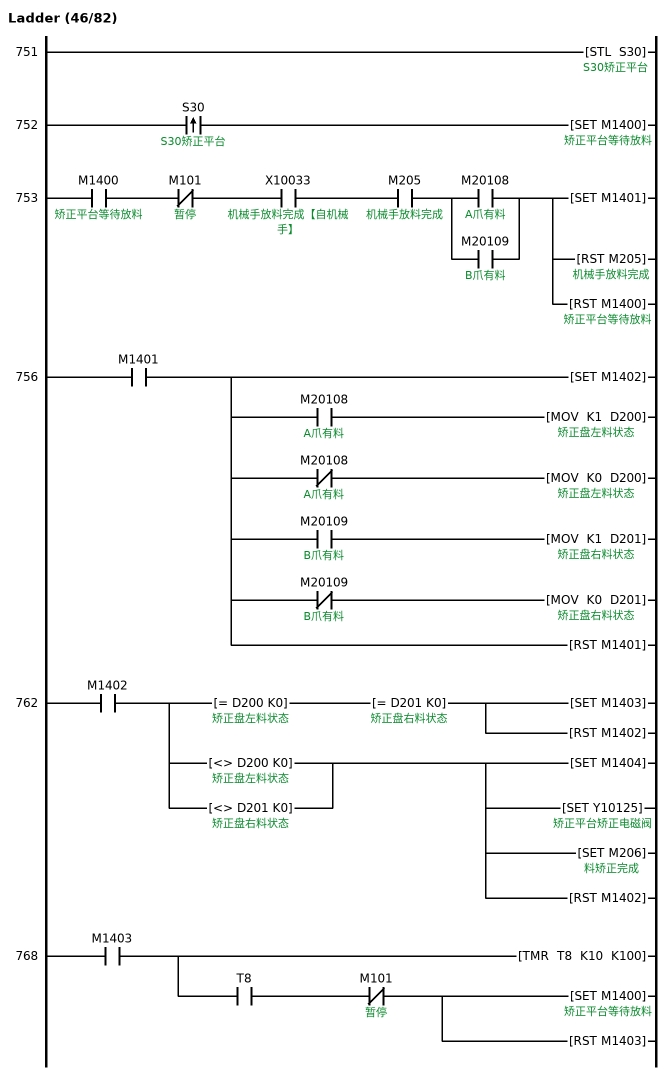
STL    S30	; S30矫正平台
LDP    S30	; S30矫正平台
SET    M1400	; 矫正平台等待放料
LD     M1400	; 矫正平台等待放料
ANI    M101	; 暂停
AND    X10033	; 机械手放料完成【自机械手】
AND    M205	; 机械手放料完成
LD     M20108	; A爪有料
OR     M20109	; B爪有料
ANB
SET    M1401
RST    M205	; 机械手放料完成
RST    M1400	; 矫正平台等待放料
LD     M1401
SET    M1402
MPS
AND    M20108	; A爪有料
MOV    K1 D200	; 矫正盘左料状态
MRD
ANI    M20108	; A爪有料
MOV    K0 D200	; 矫正盘左料状态
MRD
AND    M20109	; B爪有料
MOV    K1 D201	; 矫正盘右料状态
MRD
ANI    M20109	; B爪有料
MOV    K0 D201	; 矫正盘右料状态
MPP
RST    M1401
LD     M1402
MPS
AND=   D200 K0	; 矫正盘左料状态
AND=   D201 K0	; 矫正盘右料状态
SET    M1403
RST    M1402
MPP
LD<>   D200 K0	; 矫正盘左料状态
OR<>   D201 K0	; 矫正盘右料状态
ANB
SET    M1404
SET    Y10125	; 矫正平台矫正电磁阀
SET    M206	; 料矫正完成
RST    M1402
LD     M1403
TMR    T8 K10 K100
AND    T8
ANI    M101	; 暂停
SET    M1400	; 矫正平台等待放料
RST    M1403

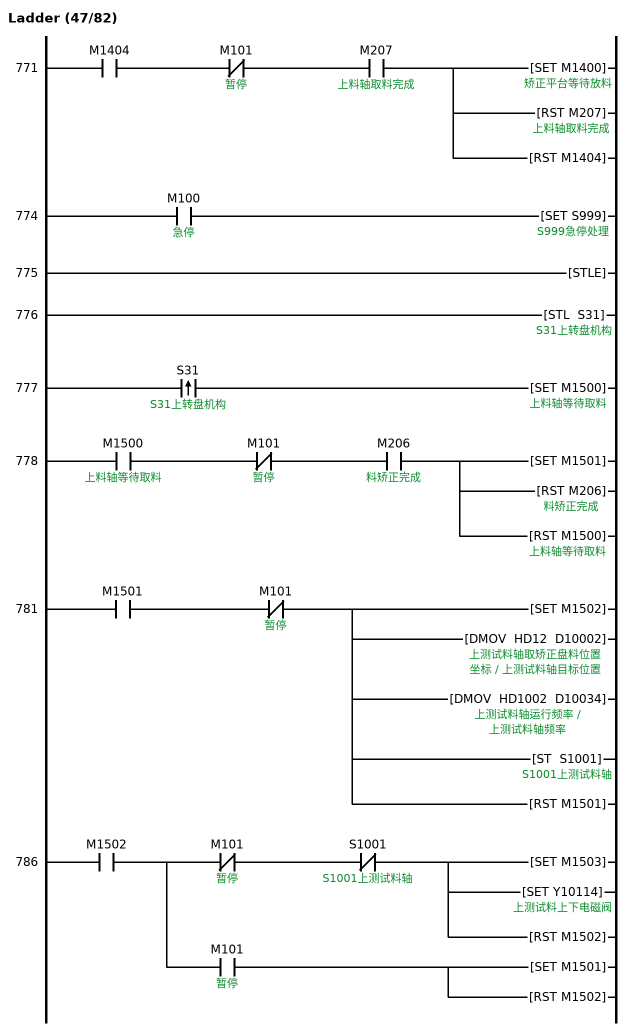
LD     M1404
ANI    M101	; 暂停
AND    M207	; 上料轴取料完成
SET    M1400	; 矫正平台等待放料
RST    M207	; 上料轴取料完成
RST    M1404
LD     M100	; 急停
SET    S999	; S999急停处理
STLE
STL    S31	; S31上转盘机构
LDP    S31	; S31上转盘机构
SET    M1500	; 上料轴等待取料
LD     M1500	; 上料轴等待取料
ANI    M101	; 暂停
AND    M206	; 料矫正完成
SET    M1501
RST    M206	; 料矫正完成
RST    M1500	; 上料轴等待取料
LD     M1501
ANI    M101	; 暂停
SET    M1502
DMOV   HD12 D10002	; 上测试料轴取矫正盘料位置坐标 / 上测试料轴目标位置
DMOV   HD1002 D10034	; 上测试料轴运行频率 / 上测试料轴频率
ST     S1001	; S1001上测试料轴
RST    M1501
LD     M1502
MPS
ANI    M101	; 暂停
ANI    S1001	; S1001上测试料轴
SET    M1503
SET    Y10114	; 上测试料上下电磁阀
RST    M1502
MPP
AND    M101	; 暂停
SET    M1501
RST    M1502

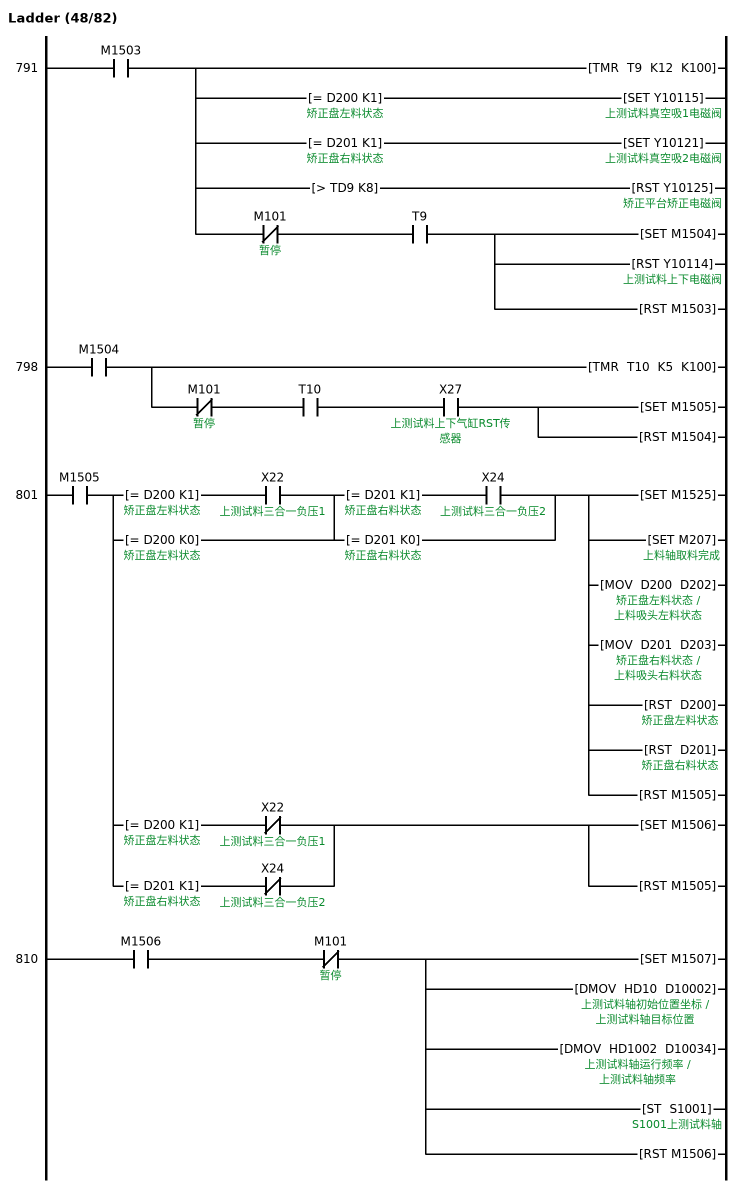
LD     M1503
TMR    T9 K12 K100
MPS
AND=   D200 K1	; 矫正盘左料状态
SET    Y10115	; 上测试料真空吸1电磁阀
MRD
AND=   D201 K1	; 矫正盘右料状态
SET    Y10121	; 上测试料真空吸2电磁阀
MRD
AND>   TD9 K8
RST    Y10125	; 矫正平台矫正电磁阀
MPP
ANI    M101	; 暂停
AND    T9
SET    M1504
RST    Y10114	; 上测试料上下电磁阀
RST    M1503
LD     M1504
TMR    T10 K5 K100
ANI    M101	; 暂停
AND    T10
AND    X27	; 上测试料上下气缸RST传感器
SET    M1505
RST    M1504
LD     M1505
MPS
LD=    D200 K1	; 矫正盘左料状态
AND    X22	; 上测试料三合一负压1
OR=    D200 K0	; 矫正盘左料状态
ANB
LD=    D201 K1	; 矫正盘右料状态
AND    X24	; 上测试料三合一负压2
OR=    D201 K0	; 矫正盘右料状态
ANB
SET    M1525
SET    M207	; 上料轴取料完成
MOV    D200 D202	; 矫正盘左料状态 / 上料吸头左料状态
MOV    D201 D203	; 矫正盘右料状态 / 上料吸头右料状态
RST    D200	; 矫正盘左料状态
RST    D201	; 矫正盘右料状态
RST    M1505
MPP
LD=    D200 K1	; 矫正盘左料状态
ANI    X22	; 上测试料三合一负压1
LD=    D201 K1	; 矫正盘右料状态
ANI    X24	; 上测试料三合一负压2
ORB
ANB
SET    M1506
RST    M1505
LD     M1506
ANI    M101	; 暂停
SET    M1507
DMOV   HD10 D10002	; 上测试料轴初始位置坐标 / 上测试料轴目标位置
DMOV   HD1002 D10034	; 上测试料轴运行频率 / 上测试料轴频率
ST     S1001	; S1001上测试料轴
RST    M1506

